Yaskawa INFORM job: SEQUENCE69.JBI

/JOB
//NAME SEQUENCE69
///FOLDERNAME INNE
//POS
///NPOS 1,1,0,0,0,0
///TOOL 0
///POSTYPE PULSE
///PULSE
C00000=42894,52348,-14453,-11880,104885,-69782
BC00000=172256,1342024,1075175
//INST
///DATE 2023/11/01 18:40
///ATTR SC,RW
///GROUP1 RB1,BS1
NOP
'Sequence69
MOVJ C00000 BC00000 VJ=100.00
END
